// TIA Portal V16 export
// export: Created 2024-09-05T17:39:15.2056473Z, ExportSetting WithDefaults, DisplayName Totally Integrated Automation Portal, DisplayVersion V16 Update 6, DisplayName TIA Portal Version Control Interface, DisplayVersion V16 Update 2, DisplayName TIA Portal Openness, DisplayVersion V16 Update 6, DisplayName STEP 7 Professional, DisplayVersion V16 Update 6, DisplayName STEP 7 Safety, DisplayVersion V16, DisplayName WinCC Advanced, DisplayVersion V16 Update 6
FUNCTION_BLOCK "ModeSelection"   // FB38, GRAPH
VERSION : 0.1
// stored: AcknowledgeErrorsRequired true, AutoNumber true, GraphVersion 6.0, InitialValuesAcquisition false, IsIECCheckEnabled false, LanguageInNetworks LAD, LockOperatingMode false, PermanentILProcessingInMANMode false, SetENOAutomatically false, SkipSteps false, UDAEnableTagReadback false, WithAlarmHandling true
   // inherited from GRAPH_BASE
   VAR
      OFF_SQ_BASE : Bool;
   END_VAR
   VAR_INPUT
      iSafetyOKauto : Bool;
      iSafetyOKmanual : Bool;
      iBasePosition : Bool;
      iPozadavekZastavitOdDveri : Bool;
      iLinkaZastavena : Bool;
      iLinkaPrazdna : Bool;
      iBaseInManualMode : Bool;
      OFF_SQ { ExternalAccessible := 'False'; ExternalVisible := 'False'; ExternalWritable := 'False'} : Bool := false;   // Turn sequence off
      INIT_SQ { ExternalAccessible := 'False'; ExternalVisible := 'False'; ExternalWritable := 'False'} : Bool := false;   // Set sequence to initial state
      ACK_EF { ExternalAccessible := 'False'; ExternalVisible := 'False'; ExternalWritable := 'False'} : Bool := false;   // Acknowledge all errors and faults
      S_PREV { ExternalAccessible := 'False'; ExternalVisible := 'False'; ExternalWritable := 'False'} : Bool := false;   // Output previous step in parameter S_NO
      S_NEXT { ExternalAccessible := 'False'; ExternalVisible := 'False'; ExternalWritable := 'False'} : Bool := false;   // Indicate next step in parameter S_NO
      SW_AUTO { ExternalAccessible := 'False'; ExternalVisible := 'False'; ExternalWritable := 'False'} : Bool := false;   // Automatic mode
      SW_TAP { ExternalAccessible := 'False'; ExternalVisible := 'False'; ExternalWritable := 'False'} : Bool := false;   // Semiautomatic/switch with transition
      SW_TOP { ExternalAccessible := 'False'; ExternalVisible := 'False'; ExternalWritable := 'False'} : Bool := false;   // Semiautomatic/ignore transition
      SW_MAN { ExternalAccessible := 'False'; ExternalVisible := 'False'; ExternalWritable := 'False'} : Bool := false;   // Manual mode
      S_SEL { ExternalAccessible := 'False'; ExternalVisible := 'False'; ExternalWritable := 'False'} : Int := 0;   // Select step to be output to S_NO
      S_ON { ExternalAccessible := 'False'; ExternalVisible := 'False'; ExternalWritable := 'False'} : Bool := false;   // Activate step indicated in S_NO
      S_OFF { ExternalAccessible := 'False'; ExternalVisible := 'False'; ExternalWritable := 'False'} : Bool := false;   // Deactivate step indicated S_NO
      T_PUSH { ExternalAccessible := 'False'; ExternalVisible := 'False'; ExternalWritable := 'False'} : Bool := false;   // Enable transition to switch in semi automatic mode
   END_VAR
   VAR_OUTPUT
      S_NO { ExternalAccessible := 'False'; ExternalVisible := 'False'; ExternalWritable := 'False'} : Int := 0;   // Step number
      S_MORE { ExternalAccessible := 'False'; ExternalVisible := 'False'; ExternalWritable := 'False'} : Bool := false;   // More steps are available and can be shown in S_NO
      S_ACTIVE { ExternalAccessible := 'False'; ExternalVisible := 'False'; ExternalWritable := 'False'} : Bool := false;   // Step indicated in S_NO is active
      ERR_FLT { ExternalAccessible := 'False'; ExternalVisible := 'False'; ExternalWritable := 'False'} : Bool := false;   // Interlock or supervision group error
      AUTO_ON { ExternalAccessible := 'False'; ExternalVisible := 'False'; ExternalWritable := 'False'} : Bool := false;   // Automatic mode is active
      TAP_ON { ExternalAccessible := 'False'; ExternalVisible := 'False'; ExternalWritable := 'False'} : Bool := false;   // Semiautomatic mode/step with transition enabled
      TOP_ON { ExternalAccessible := 'False'; ExternalVisible := 'False'; ExternalWritable := 'False'} : Bool := false;   // Semiautomatic mode/ignore transition enabled
      MAN_ON { ExternalAccessible := 'False'; ExternalVisible := 'False'; ExternalWritable := 'False'} : Bool := false;   // Manual mode is active
   END_VAR
   VAR
      dummy : Bool;
   END_VAR
   VAR RETAIN
      mode : "udtModes";
   END_VAR
   VAR
      PrevMode : Int;
      F_TRIG_semiauto_switch { S7_SetPoint := 'True'} : F_TRIG;
      F_TRIG_switchAuto { S7_SetPoint := 'True'} : F_TRIG;
   END_VAR
BEGIN
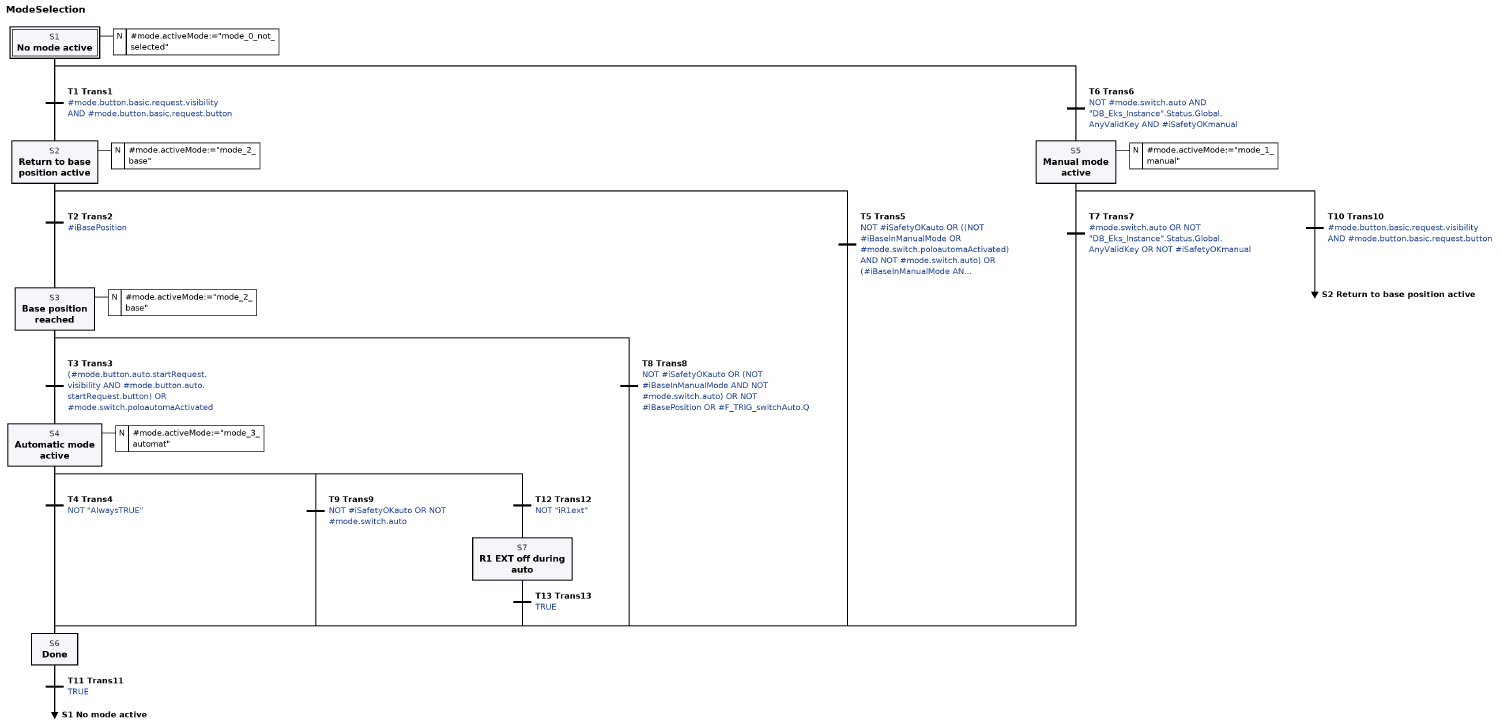
   // permanent pre-instructions
   NETWORK 1
   TITLE = mode init
      "ModeSelection_DB".mode.activeMode := "mode_0_not_selected";
   NETWORK 2
   TITLE = button visibility
      #mode.button.basic.request.visibility := #iSafetyOKauto AND ((#mode.switch.auto AND #"No mode active".X AND (NOT #iBaseInManualMode OR #mode.switch.poloautomaActivated)) OR (NOT #mode.switch.auto AND #"Manual mode active".X AND #iBaseInManualMode AND NOT #mode.switch.poloautomaActivated));
      #mode.button.auto.startRequest.visibility := #iSafetyOKauto AND #mode.switch.auto AND #"Base position reached".X AND NOT "SystemHMI".AlarmActive;
   NETWORK 3
   TITLE = semiauto switch off detection
      #F_TRIG_semiauto_switch(CLK := #mode.switch.poloautomaActivated);   // F_TRIG
   NETWORK 4
      #F_TRIG_switchAuto(CLK := #mode.switch.auto);   // F_TRIG

   // sequencer 1
   INITIAL_STEP "No mode active":   // S1, max time T#10S, warning time T#7S
              N    #mode.activeMode:="mode_0_not_selected"
   END_STEP
   TRANSITION Trans1 FROM "No mode active" TO "Return to base position active"   // T1
      := #mode.button.basic.request.visibility AND #mode.button.basic.request.button;
   END_TRANSITION
   TRANSITION Trans6 FROM "No mode active" TO "Manual mode active"   // T6
      := NOT #mode.switch.auto AND "DB_Eks_Instance".Status.Global.AnyValidKey AND #iSafetyOKmanual;
   END_TRANSITION
   STEP "Return to base position active":   // S2, max time T#10S, warning time T#7S
              N    #mode.activeMode:="mode_2_base"
   END_STEP
   TRANSITION Trans2 FROM "Return to base position active" TO "Base position reached"   // T2
      := #iBasePosition;
   END_TRANSITION
   TRANSITION Trans5 FROM "Return to base position active" TO Done   // T5
      := NOT #iSafetyOKauto OR ((NOT #iBaseInManualMode OR #mode.switch.poloautomaActivated) AND NOT #mode.switch.auto) OR (#iBaseInManualMode AND #mode.switch.auto AND NOT #mode.switch.poloautomaActivated) OR #F_TRIG_semiauto_switch.Q;
   END_TRANSITION
   STEP "Base position reached":   // S3, max time T#10S, warning time T#7S
              N    #mode.activeMode:="mode_2_base"
   END_STEP
   TRANSITION Trans3 FROM "Base position reached" TO "Automatic mode active"   // T3
      := (#mode.button.auto.startRequest.visibility AND #mode.button.auto.startRequest.button) OR #mode.switch.poloautomaActivated;
   END_TRANSITION
   TRANSITION Trans8 FROM "Base position reached" TO Done   // T8
      := NOT #iSafetyOKauto OR (NOT #iBaseInManualMode AND NOT #mode.switch.auto) OR NOT #iBasePosition OR #F_TRIG_switchAuto.Q;
   END_TRANSITION
   STEP "Automatic mode active":   // S4, max time T#10S, warning time T#7S
              N    #mode.activeMode:="mode_3_automat"
   END_STEP
   TRANSITION Trans4 FROM "Automatic mode active" TO Done   // T4
      := NOT "AlwaysTRUE";
   END_TRANSITION
   TRANSITION Trans9 FROM "Automatic mode active" TO Done   // T9
      := NOT #iSafetyOKauto OR NOT #mode.switch.auto;
   END_TRANSITION
   TRANSITION Trans12 FROM "Automatic mode active" TO "R1 EXT off during auto"   // T12
      := NOT "iR1ext";
   END_TRANSITION
   STEP "Manual mode active":   // S5, max time T#10S, warning time T#7S
              N    #mode.activeMode:="mode_1_manual"
   END_STEP
   TRANSITION Trans7 FROM "Manual mode active" TO Done   // T7
      := #mode.switch.auto OR NOT "DB_Eks_Instance".Status.Global.AnyValidKey OR NOT #iSafetyOKmanual;
   END_TRANSITION
   TRANSITION Trans10 FROM "Manual mode active" TO "Return to base position active"   // T10, jump
      := #mode.button.basic.request.visibility AND #mode.button.basic.request.button;
   END_TRANSITION
   STEP Done:   // S6, max time T#10S, warning time T#7S
   END_STEP
   TRANSITION Trans11 FROM Done TO "No mode active"   // T11, jump
      := TRUE;
   END_TRANSITION
   STEP "R1 EXT off during auto":   // S7, max time T#10S, warning time T#7S
   END_STEP
   TRANSITION Trans13 FROM "R1 EXT off during auto" TO Done   // T13
      := TRUE;
   END_TRANSITION

   // permanent post-instructions
   NETWORK 1
   TITLE = semiauto mode
      IF ((#mode.activeMode = "mode_2_base") OR (#mode.activeMode = "mode_3_automat")) AND #mode.switch.poloautomaActivated THEN
          #mode.activeMode := "mode_4_semiautomat";
      END_IF;
   NETWORK 2
   TITLE = previous mode
      #mode.modeChanged := #mode.activeMode <> #PrevMode;
      #PrevMode := #mode.activeMode;
END_FUNCTION_BLOCK
